TYPE Level_Keys_DUT :
STRUCT
	Level:	ARRAY[1..6] OF BOOL;
END_STRUCT
END_TYPE

(* stored: Version 1.1.0.1
   DUT Level_Keys_DUT: Id {1749397a-9cff-4d03-88fe-f97180a71009} *)
